// TIA Portal V20 export
TYPE "LER_zp_CITIEoC"
// stored: Access Published
   STRUCT
      PUN_Ready : Bool;   // PUN Ready
      FTQ_DataReady : Bool;   // FTQ Data Ready
      Energy_Conservation_Enable : Bool;   // Energy Conservation Enable
      Buffer_Bypassed : Bool;   // Buffer Bypassed
      Bypassed : Bool;   // Bypassed
      Safety_Checksum_OK : Bool;   // Safety Checksum OK
      Spare_7 : Bool;
      Spare_8 : Bool;
      Spare_SINT : SInt;
      Spare_INT : Int;
      PUN_Data : String[20];   // PUN Data
      FTQ_PUN_Data : String[20];   // FTQ PUN Data
      PUN_GM_Part_Num : String[8];   // PUN GM Part Number
      PUN_Optional_Data : String[12];   // PUN Optional Data
      Part_Type : String[12];   // Part Type
      Reject_Message : String[100];   // Reject Message
      AOI_Revision : Int;   // AOI Revision
      Good_Count : Int;   // Good Count
      Reject_Count : Int;   // Reject Count
      Buffer_Count : Int;   // Buffer Count
      LastLoadTime : Int;   // Last Load Time
      LastUnloadTIme : Int;   // Last Unload Time
      Part_Type_Message : Int;   // Part Type Message
      Bypassed_Pallet_Count : Int;   // Bypass Pallet Count
      Filter_Current_Temp : Int;   // Filter Current Temp
      Filter_NumQuantity_1 : Int;   // Filter Numerical Quantity 1
      Filter_NumQuantity_2 : Int;   // Filter Numerical Quantity 2
      Filter_NumQuantity_3 : Int;   // Filter Numerical Quantity 3
      Spare_INT_2 : Int;
      Rated_Cycle_Time : DInt;   // Rated Cycle Time
      Last_Cycle_Time : DInt;   // Last Cycle Time
      LastProcessingTime : DInt;   // Last Processing Time
      Reject_Code : DInt;   // Reject Code
   END_STRUCT;
END_TYPE
